// TIA Portal V17 export
// export: Created 2025-03-07T09:17:02.6439569Z, ExportSetting WithDefaults, DisplayName Totally Integrated Automation Portal, DisplayVersion V17 Update 8, DisplayName TIA Portal Openness, DisplayVersion V17 Update 8, DisplayName TIA Portal Version Control Interface, DisplayVersion V17, DisplayName SINAMICS Startdrive Advanced, DisplayVersion V17 SP2, DisplayName SINAMICS Startdrive G110M, G120, G120C, G120D, G120P, G115D, DisplayVersion V17 SP2, DisplayName SINAMICS Startdrive G130, G150, S120, S150, SINAMICS MV, S210, DisplayVersion V17 SP2, DisplayName STEP 7 Professional, DisplayVersion V17 Update 8, DisplayName SINUMERIK ONE STEP 7 Toolbox, DisplayVersion V17 Update 12, DisplayName SINUMERIK 840D sl STEP 7 Toolbox, DisplayVersion V17 Update 12, DisplayName STEP 7 Safety, DisplayVersion V17 Update 6, DisplayName WinCC Advanced, DisplayVersion V17 Update 8
FUNCTION "FC7450_QUALITY_CHECK_CLADDING" : Void   // FC7450, LAD
{ S7_Optimized_Access := 'FALSE' }
AUTHOR : ETXETAR
NAME : GM-QC
VERSION : 1.0
// stored: AutoNumber false, IsIECCheckEnabled false, SetENOAutomatically false, UDAEnableTagReadback false
BEGIN

REGION Network 1: OPTIONS OFF
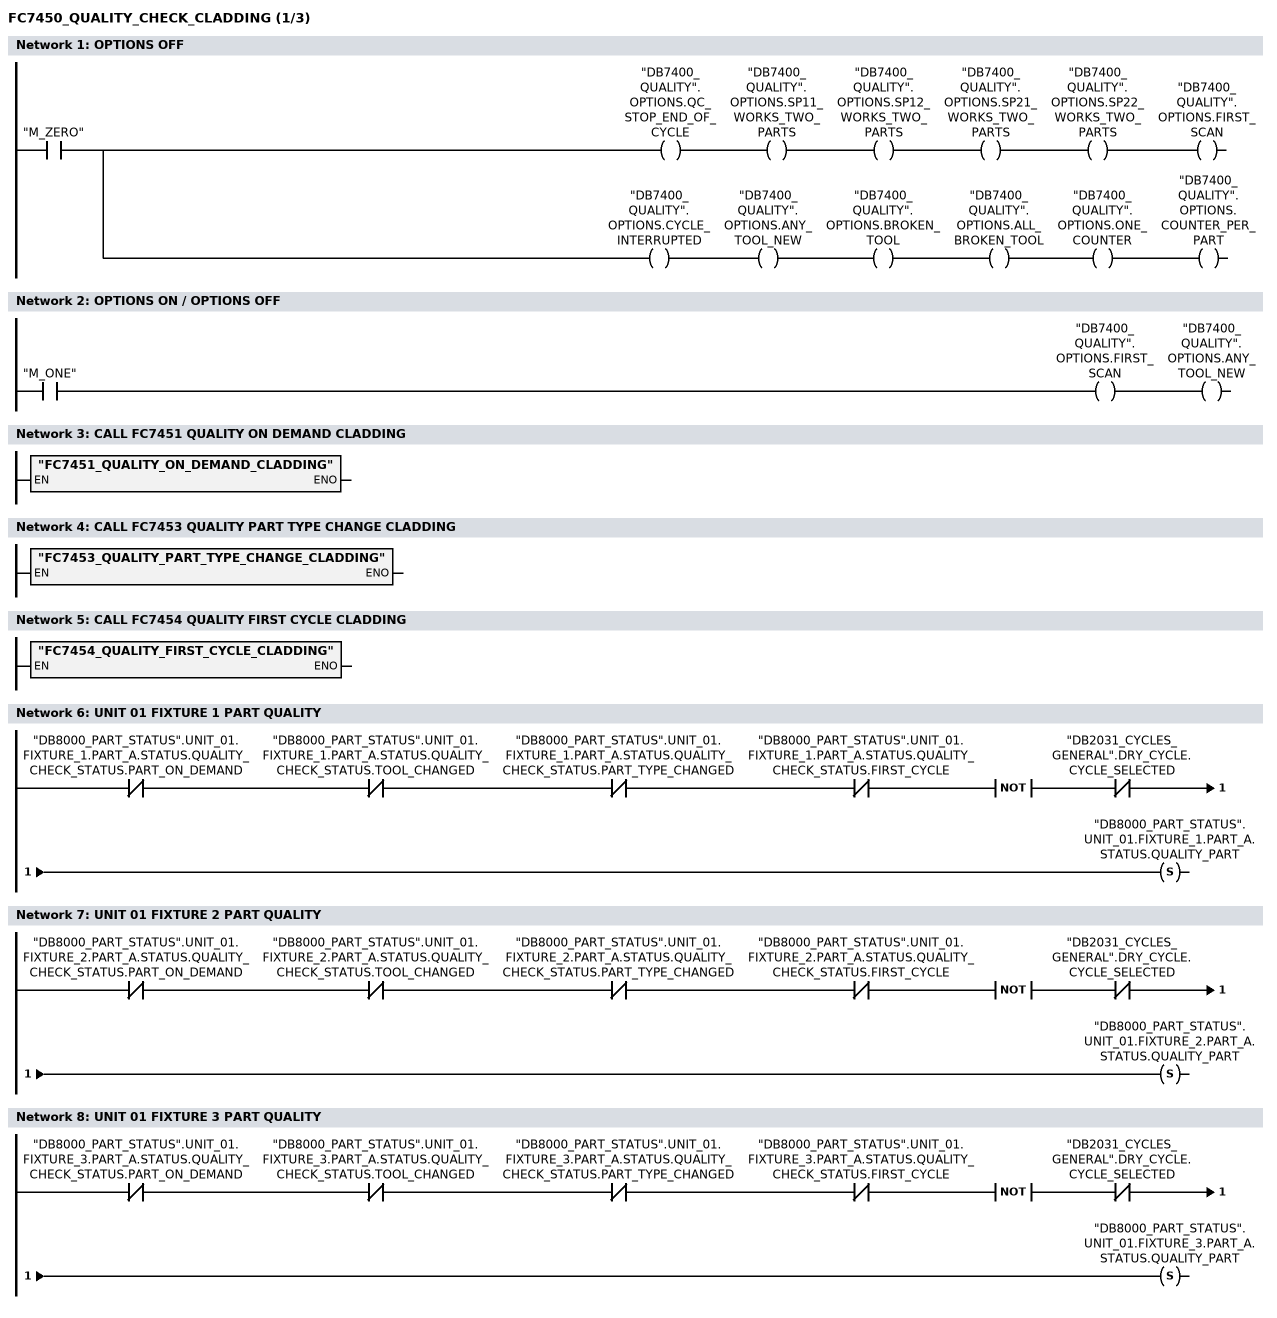
   RUNG wire#powerrail
      Contact( "M_ZERO" )
      wire#w1
      Coil( "DB7400_QUALITY".OPTIONS.QC_STOP_END_OF_CYCLE )
      Coil( "DB7400_QUALITY".OPTIONS.SP11_WORKS_TWO_PARTS )
      Coil( "DB7400_QUALITY".OPTIONS.SP12_WORKS_TWO_PARTS )
      Coil( "DB7400_QUALITY".OPTIONS.SP21_WORKS_TWO_PARTS )
      Coil( "DB7400_QUALITY".OPTIONS.SP22_WORKS_TWO_PARTS )
      Coil( "DB7400_QUALITY".OPTIONS.FIRST_SCAN )
   END_RUNG
   RUNG wire#w1
      Coil( "DB7400_QUALITY".OPTIONS.CYCLE_INTERRUPTED )
      Coil( "DB7400_QUALITY".OPTIONS.ANY_TOOL_NEW )
      Coil( "DB7400_QUALITY".OPTIONS.BROKEN_TOOL )
      Coil( "DB7400_QUALITY".OPTIONS.ALL_BROKEN_TOOL )
      Coil( "DB7400_QUALITY".OPTIONS.ONE_COUNTER )
      Coil( "DB7400_QUALITY".OPTIONS.COUNTER_PER_PART )
   END_RUNG
   // the same network as SCL:
   "DB7400_QUALITY".OPTIONS.QC_STOP_END_OF_CYCLE := "M_ZERO";
   "DB7400_QUALITY".OPTIONS.SP11_WORKS_TWO_PARTS := "M_ZERO";
   "DB7400_QUALITY".OPTIONS.SP12_WORKS_TWO_PARTS := "M_ZERO";
   "DB7400_QUALITY".OPTIONS.SP21_WORKS_TWO_PARTS := "M_ZERO";
   "DB7400_QUALITY".OPTIONS.SP22_WORKS_TWO_PARTS := "M_ZERO";
   "DB7400_QUALITY".OPTIONS.FIRST_SCAN := "M_ZERO";
   "DB7400_QUALITY".OPTIONS.CYCLE_INTERRUPTED := "M_ZERO";
   "DB7400_QUALITY".OPTIONS.ANY_TOOL_NEW := "M_ZERO";
   "DB7400_QUALITY".OPTIONS.BROKEN_TOOL := "M_ZERO";
   "DB7400_QUALITY".OPTIONS.ALL_BROKEN_TOOL := "M_ZERO";
   "DB7400_QUALITY".OPTIONS.ONE_COUNTER := "M_ZERO";
   "DB7400_QUALITY".OPTIONS.COUNTER_PER_PART := "M_ZERO";
END_REGION

REGION Network 2: OPTIONS ON / OPTIONS OFF
   RUNG wire#powerrail
      Contact( "M_ONE" )
      Coil( "DB7400_QUALITY".OPTIONS.FIRST_SCAN )
      Coil( "DB7400_QUALITY".OPTIONS.ANY_TOOL_NEW )
   END_RUNG
   // the same network as SCL:
   "DB7400_QUALITY".OPTIONS.FIRST_SCAN := "M_ONE";
   "DB7400_QUALITY".OPTIONS.ANY_TOOL_NEW := "M_ONE";
END_REGION

REGION Network 3: CALL FC7451 QUALITY ON DEMAND CLADDING
   RUNG wire#powerrail
      "FC7451_QUALITY_ON_DEMAND_CLADDING"()
   END_RUNG
   // the same network as SCL:
   "FC7451_QUALITY_ON_DEMAND_CLADDING"();
END_REGION

REGION Network 4: CALL FC7453 QUALITY PART TYPE CHANGE CLADDING
   RUNG wire#powerrail
      "FC7453_QUALITY_PART_TYPE_CHANGE_CLADDING"()
   END_RUNG
   // the same network as SCL:
   "FC7453_QUALITY_PART_TYPE_CHANGE_CLADDING"();
END_REGION

REGION Network 5: CALL FC7454 QUALITY FIRST CYCLE CLADDING
   RUNG wire#powerrail
      "FC7454_QUALITY_FIRST_CYCLE_CLADDING"()
   END_RUNG
   // the same network as SCL:
   "FC7454_QUALITY_FIRST_CYCLE_CLADDING"();
END_REGION

REGION Network 6: UNIT 01 FIXTURE 1 PART QUALITY
   RUNG wire#powerrail
      I_Contact( "DB8000_PART_STATUS".UNIT_01.FIXTURE_1.PART_A.STATUS.QUALITY_CHECK_STATUS.PART_ON_DEMAND )
      I_Contact( "DB8000_PART_STATUS".UNIT_01.FIXTURE_1.PART_A.STATUS.QUALITY_CHECK_STATUS.TOOL_CHANGED )
      I_Contact( "DB8000_PART_STATUS".UNIT_01.FIXTURE_1.PART_A.STATUS.QUALITY_CHECK_STATUS.PART_TYPE_CHANGED )
      I_Contact( "DB8000_PART_STATUS".UNIT_01.FIXTURE_1.PART_A.STATUS.QUALITY_CHECK_STATUS.FIRST_CYCLE )
      Not()
      I_Contact( "DB2031_CYCLES_GENERAL".DRY_CYCLE.CYCLE_SELECTED )
      S_Coil( "DB8000_PART_STATUS".UNIT_01.FIXTURE_1.PART_A.STATUS.QUALITY_PART )
   END_RUNG
   // the same network as SCL:
   IF NOT (NOT "DB8000_PART_STATUS".UNIT_01.FIXTURE_1.PART_A.STATUS.QUALITY_CHECK_STATUS.PART_ON_DEMAND AND NOT "DB8000_PART_STATUS".UNIT_01.FIXTURE_1.PART_A.STATUS.QUALITY_CHECK_STATUS.TOOL_CHANGED AND NOT "DB8000_PART_STATUS".UNIT_01.FIXTURE_1.PART_A.STATUS.QUALITY_CHECK_STATUS.PART_TYPE_CHANGED AND NOT "DB8000_PART_STATUS".UNIT_01.FIXTURE_1.PART_A.STATUS.QUALITY_CHECK_STATUS.FIRST_CYCLE) AND NOT "DB2031_CYCLES_GENERAL".DRY_CYCLE.CYCLE_SELECTED THEN
       "DB8000_PART_STATUS".UNIT_01.FIXTURE_1.PART_A.STATUS.QUALITY_PART := TRUE;
   END_IF;
END_REGION

REGION Network 7: UNIT 01 FIXTURE 2 PART QUALITY
   RUNG wire#powerrail
      I_Contact( "DB8000_PART_STATUS".UNIT_01.FIXTURE_2.PART_A.STATUS.QUALITY_CHECK_STATUS.PART_ON_DEMAND )
      I_Contact( "DB8000_PART_STATUS".UNIT_01.FIXTURE_2.PART_A.STATUS.QUALITY_CHECK_STATUS.TOOL_CHANGED )
      I_Contact( "DB8000_PART_STATUS".UNIT_01.FIXTURE_2.PART_A.STATUS.QUALITY_CHECK_STATUS.PART_TYPE_CHANGED )
      I_Contact( "DB8000_PART_STATUS".UNIT_01.FIXTURE_2.PART_A.STATUS.QUALITY_CHECK_STATUS.FIRST_CYCLE )
      Not()
      I_Contact( "DB2031_CYCLES_GENERAL".DRY_CYCLE.CYCLE_SELECTED )
      S_Coil( "DB8000_PART_STATUS".UNIT_01.FIXTURE_2.PART_A.STATUS.QUALITY_PART )
   END_RUNG
   // the same network as SCL:
   IF NOT (NOT "DB8000_PART_STATUS".UNIT_01.FIXTURE_2.PART_A.STATUS.QUALITY_CHECK_STATUS.PART_ON_DEMAND AND NOT "DB8000_PART_STATUS".UNIT_01.FIXTURE_2.PART_A.STATUS.QUALITY_CHECK_STATUS.TOOL_CHANGED AND NOT "DB8000_PART_STATUS".UNIT_01.FIXTURE_2.PART_A.STATUS.QUALITY_CHECK_STATUS.PART_TYPE_CHANGED AND NOT "DB8000_PART_STATUS".UNIT_01.FIXTURE_2.PART_A.STATUS.QUALITY_CHECK_STATUS.FIRST_CYCLE) AND NOT "DB2031_CYCLES_GENERAL".DRY_CYCLE.CYCLE_SELECTED THEN
       "DB8000_PART_STATUS".UNIT_01.FIXTURE_2.PART_A.STATUS.QUALITY_PART := TRUE;
   END_IF;
END_REGION

REGION Network 8: UNIT 01 FIXTURE 3 PART QUALITY
   RUNG wire#powerrail
      I_Contact( "DB8000_PART_STATUS".UNIT_01.FIXTURE_3.PART_A.STATUS.QUALITY_CHECK_STATUS.PART_ON_DEMAND )
      I_Contact( "DB8000_PART_STATUS".UNIT_01.FIXTURE_3.PART_A.STATUS.QUALITY_CHECK_STATUS.TOOL_CHANGED )
      I_Contact( "DB8000_PART_STATUS".UNIT_01.FIXTURE_3.PART_A.STATUS.QUALITY_CHECK_STATUS.PART_TYPE_CHANGED )
      I_Contact( "DB8000_PART_STATUS".UNIT_01.FIXTURE_3.PART_A.STATUS.QUALITY_CHECK_STATUS.FIRST_CYCLE )
      Not()
      I_Contact( "DB2031_CYCLES_GENERAL".DRY_CYCLE.CYCLE_SELECTED )
      S_Coil( "DB8000_PART_STATUS".UNIT_01.FIXTURE_3.PART_A.STATUS.QUALITY_PART )
   END_RUNG
   // the same network as SCL:
   IF NOT (NOT "DB8000_PART_STATUS".UNIT_01.FIXTURE_3.PART_A.STATUS.QUALITY_CHECK_STATUS.PART_ON_DEMAND AND NOT "DB8000_PART_STATUS".UNIT_01.FIXTURE_3.PART_A.STATUS.QUALITY_CHECK_STATUS.TOOL_CHANGED AND NOT "DB8000_PART_STATUS".UNIT_01.FIXTURE_3.PART_A.STATUS.QUALITY_CHECK_STATUS.PART_TYPE_CHANGED AND NOT "DB8000_PART_STATUS".UNIT_01.FIXTURE_3.PART_A.STATUS.QUALITY_CHECK_STATUS.FIRST_CYCLE) AND NOT "DB2031_CYCLES_GENERAL".DRY_CYCLE.CYCLE_SELECTED THEN
       "DB8000_PART_STATUS".UNIT_01.FIXTURE_3.PART_A.STATUS.QUALITY_PART := TRUE;
   END_IF;
END_REGION

REGION Network 9: UNIT 01 FIXTURE 4 PART QUALITY
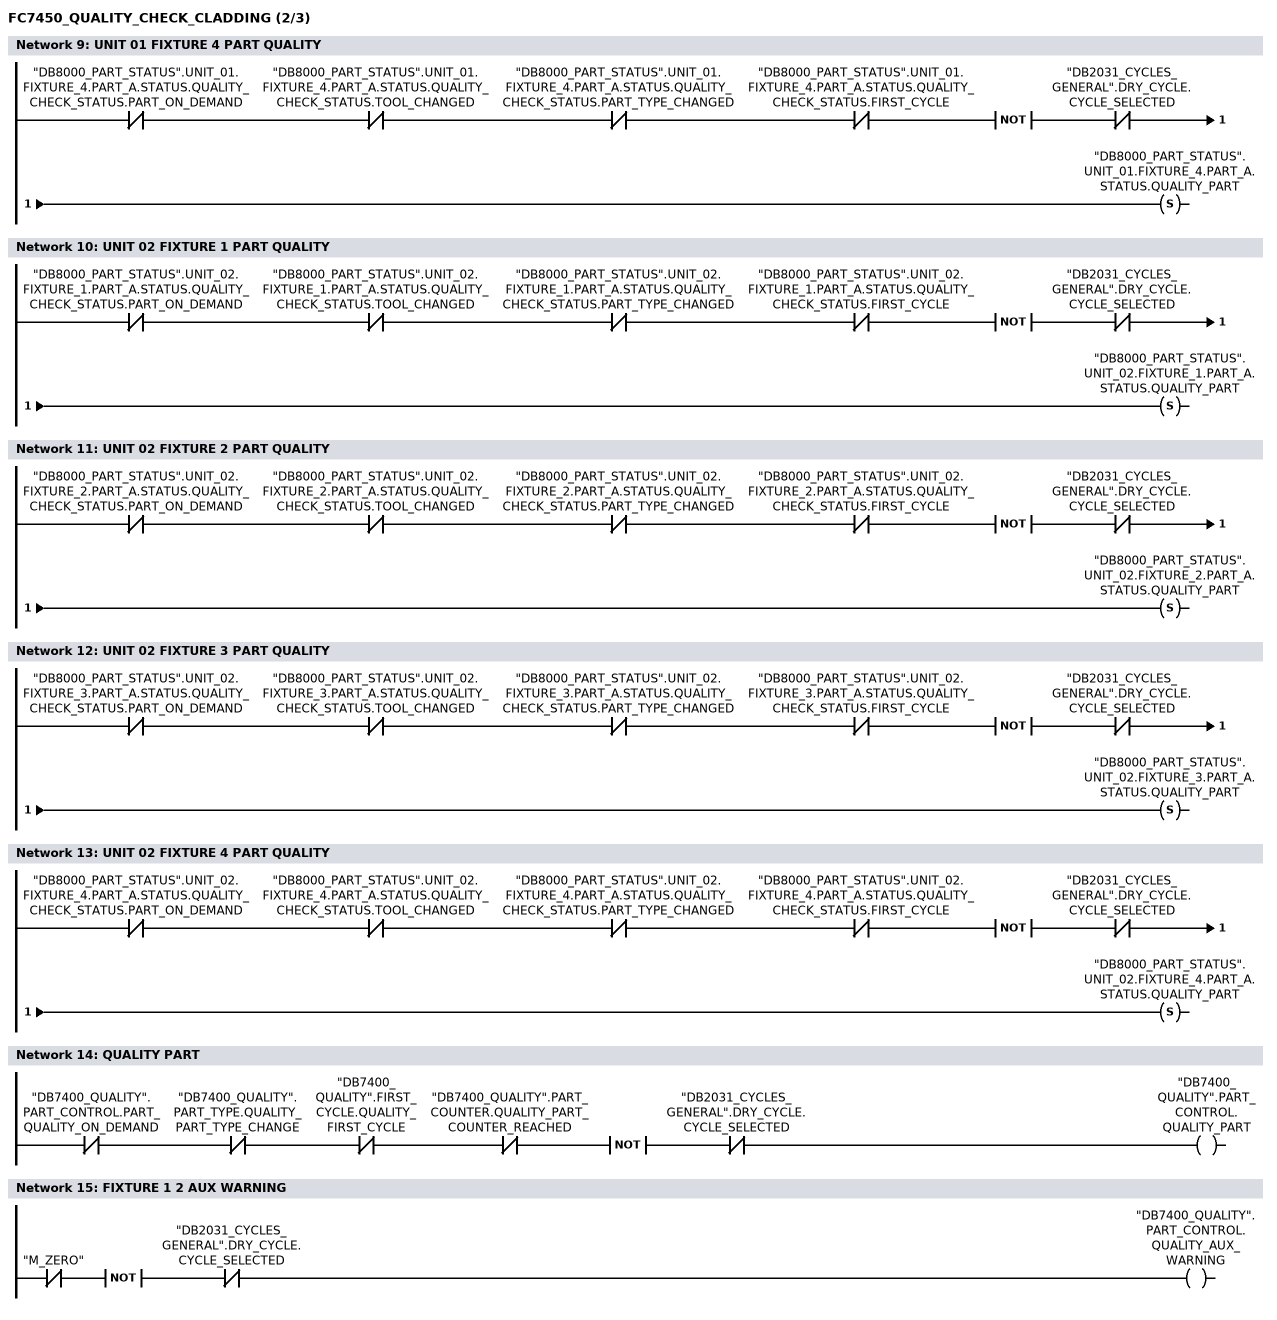
   RUNG wire#powerrail
      I_Contact( "DB8000_PART_STATUS".UNIT_01.FIXTURE_4.PART_A.STATUS.QUALITY_CHECK_STATUS.PART_ON_DEMAND )
      I_Contact( "DB8000_PART_STATUS".UNIT_01.FIXTURE_4.PART_A.STATUS.QUALITY_CHECK_STATUS.TOOL_CHANGED )
      I_Contact( "DB8000_PART_STATUS".UNIT_01.FIXTURE_4.PART_A.STATUS.QUALITY_CHECK_STATUS.PART_TYPE_CHANGED )
      I_Contact( "DB8000_PART_STATUS".UNIT_01.FIXTURE_4.PART_A.STATUS.QUALITY_CHECK_STATUS.FIRST_CYCLE )
      Not()
      I_Contact( "DB2031_CYCLES_GENERAL".DRY_CYCLE.CYCLE_SELECTED )
      S_Coil( "DB8000_PART_STATUS".UNIT_01.FIXTURE_4.PART_A.STATUS.QUALITY_PART )
   END_RUNG
   // the same network as SCL:
   IF NOT (NOT "DB8000_PART_STATUS".UNIT_01.FIXTURE_4.PART_A.STATUS.QUALITY_CHECK_STATUS.PART_ON_DEMAND AND NOT "DB8000_PART_STATUS".UNIT_01.FIXTURE_4.PART_A.STATUS.QUALITY_CHECK_STATUS.TOOL_CHANGED AND NOT "DB8000_PART_STATUS".UNIT_01.FIXTURE_4.PART_A.STATUS.QUALITY_CHECK_STATUS.PART_TYPE_CHANGED AND NOT "DB8000_PART_STATUS".UNIT_01.FIXTURE_4.PART_A.STATUS.QUALITY_CHECK_STATUS.FIRST_CYCLE) AND NOT "DB2031_CYCLES_GENERAL".DRY_CYCLE.CYCLE_SELECTED THEN
       "DB8000_PART_STATUS".UNIT_01.FIXTURE_4.PART_A.STATUS.QUALITY_PART := TRUE;
   END_IF;
END_REGION

REGION Network 10: UNIT 02 FIXTURE 1 PART QUALITY
   RUNG wire#powerrail
      I_Contact( "DB8000_PART_STATUS".UNIT_02.FIXTURE_1.PART_A.STATUS.QUALITY_CHECK_STATUS.PART_ON_DEMAND )
      I_Contact( "DB8000_PART_STATUS".UNIT_02.FIXTURE_1.PART_A.STATUS.QUALITY_CHECK_STATUS.TOOL_CHANGED )
      I_Contact( "DB8000_PART_STATUS".UNIT_02.FIXTURE_1.PART_A.STATUS.QUALITY_CHECK_STATUS.PART_TYPE_CHANGED )
      I_Contact( "DB8000_PART_STATUS".UNIT_02.FIXTURE_1.PART_A.STATUS.QUALITY_CHECK_STATUS.FIRST_CYCLE )
      Not()
      I_Contact( "DB2031_CYCLES_GENERAL".DRY_CYCLE.CYCLE_SELECTED )
      S_Coil( "DB8000_PART_STATUS".UNIT_02.FIXTURE_1.PART_A.STATUS.QUALITY_PART )
   END_RUNG
   // the same network as SCL:
   IF NOT (NOT "DB8000_PART_STATUS".UNIT_02.FIXTURE_1.PART_A.STATUS.QUALITY_CHECK_STATUS.PART_ON_DEMAND AND NOT "DB8000_PART_STATUS".UNIT_02.FIXTURE_1.PART_A.STATUS.QUALITY_CHECK_STATUS.TOOL_CHANGED AND NOT "DB8000_PART_STATUS".UNIT_02.FIXTURE_1.PART_A.STATUS.QUALITY_CHECK_STATUS.PART_TYPE_CHANGED AND NOT "DB8000_PART_STATUS".UNIT_02.FIXTURE_1.PART_A.STATUS.QUALITY_CHECK_STATUS.FIRST_CYCLE) AND NOT "DB2031_CYCLES_GENERAL".DRY_CYCLE.CYCLE_SELECTED THEN
       "DB8000_PART_STATUS".UNIT_02.FIXTURE_1.PART_A.STATUS.QUALITY_PART := TRUE;
   END_IF;
END_REGION

REGION Network 11: UNIT 02 FIXTURE 2 PART QUALITY
   RUNG wire#powerrail
      I_Contact( "DB8000_PART_STATUS".UNIT_02.FIXTURE_2.PART_A.STATUS.QUALITY_CHECK_STATUS.PART_ON_DEMAND )
      I_Contact( "DB8000_PART_STATUS".UNIT_02.FIXTURE_2.PART_A.STATUS.QUALITY_CHECK_STATUS.TOOL_CHANGED )
      I_Contact( "DB8000_PART_STATUS".UNIT_02.FIXTURE_2.PART_A.STATUS.QUALITY_CHECK_STATUS.PART_TYPE_CHANGED )
      I_Contact( "DB8000_PART_STATUS".UNIT_02.FIXTURE_2.PART_A.STATUS.QUALITY_CHECK_STATUS.FIRST_CYCLE )
      Not()
      I_Contact( "DB2031_CYCLES_GENERAL".DRY_CYCLE.CYCLE_SELECTED )
      S_Coil( "DB8000_PART_STATUS".UNIT_02.FIXTURE_2.PART_A.STATUS.QUALITY_PART )
   END_RUNG
   // the same network as SCL:
   IF NOT (NOT "DB8000_PART_STATUS".UNIT_02.FIXTURE_2.PART_A.STATUS.QUALITY_CHECK_STATUS.PART_ON_DEMAND AND NOT "DB8000_PART_STATUS".UNIT_02.FIXTURE_2.PART_A.STATUS.QUALITY_CHECK_STATUS.TOOL_CHANGED AND NOT "DB8000_PART_STATUS".UNIT_02.FIXTURE_2.PART_A.STATUS.QUALITY_CHECK_STATUS.PART_TYPE_CHANGED AND NOT "DB8000_PART_STATUS".UNIT_02.FIXTURE_2.PART_A.STATUS.QUALITY_CHECK_STATUS.FIRST_CYCLE) AND NOT "DB2031_CYCLES_GENERAL".DRY_CYCLE.CYCLE_SELECTED THEN
       "DB8000_PART_STATUS".UNIT_02.FIXTURE_2.PART_A.STATUS.QUALITY_PART := TRUE;
   END_IF;
END_REGION

REGION Network 12: UNIT 02 FIXTURE 3 PART QUALITY
   RUNG wire#powerrail
      I_Contact( "DB8000_PART_STATUS".UNIT_02.FIXTURE_3.PART_A.STATUS.QUALITY_CHECK_STATUS.PART_ON_DEMAND )
      I_Contact( "DB8000_PART_STATUS".UNIT_02.FIXTURE_3.PART_A.STATUS.QUALITY_CHECK_STATUS.TOOL_CHANGED )
      I_Contact( "DB8000_PART_STATUS".UNIT_02.FIXTURE_3.PART_A.STATUS.QUALITY_CHECK_STATUS.PART_TYPE_CHANGED )
      I_Contact( "DB8000_PART_STATUS".UNIT_02.FIXTURE_3.PART_A.STATUS.QUALITY_CHECK_STATUS.FIRST_CYCLE )
      Not()
      I_Contact( "DB2031_CYCLES_GENERAL".DRY_CYCLE.CYCLE_SELECTED )
      S_Coil( "DB8000_PART_STATUS".UNIT_02.FIXTURE_3.PART_A.STATUS.QUALITY_PART )
   END_RUNG
   // the same network as SCL:
   IF NOT (NOT "DB8000_PART_STATUS".UNIT_02.FIXTURE_3.PART_A.STATUS.QUALITY_CHECK_STATUS.PART_ON_DEMAND AND NOT "DB8000_PART_STATUS".UNIT_02.FIXTURE_3.PART_A.STATUS.QUALITY_CHECK_STATUS.TOOL_CHANGED AND NOT "DB8000_PART_STATUS".UNIT_02.FIXTURE_3.PART_A.STATUS.QUALITY_CHECK_STATUS.PART_TYPE_CHANGED AND NOT "DB8000_PART_STATUS".UNIT_02.FIXTURE_3.PART_A.STATUS.QUALITY_CHECK_STATUS.FIRST_CYCLE) AND NOT "DB2031_CYCLES_GENERAL".DRY_CYCLE.CYCLE_SELECTED THEN
       "DB8000_PART_STATUS".UNIT_02.FIXTURE_3.PART_A.STATUS.QUALITY_PART := TRUE;
   END_IF;
END_REGION

REGION Network 13: UNIT 02 FIXTURE 4 PART QUALITY
   RUNG wire#powerrail
      I_Contact( "DB8000_PART_STATUS".UNIT_02.FIXTURE_4.PART_A.STATUS.QUALITY_CHECK_STATUS.PART_ON_DEMAND )
      I_Contact( "DB8000_PART_STATUS".UNIT_02.FIXTURE_4.PART_A.STATUS.QUALITY_CHECK_STATUS.TOOL_CHANGED )
      I_Contact( "DB8000_PART_STATUS".UNIT_02.FIXTURE_4.PART_A.STATUS.QUALITY_CHECK_STATUS.PART_TYPE_CHANGED )
      I_Contact( "DB8000_PART_STATUS".UNIT_02.FIXTURE_4.PART_A.STATUS.QUALITY_CHECK_STATUS.FIRST_CYCLE )
      Not()
      I_Contact( "DB2031_CYCLES_GENERAL".DRY_CYCLE.CYCLE_SELECTED )
      S_Coil( "DB8000_PART_STATUS".UNIT_02.FIXTURE_4.PART_A.STATUS.QUALITY_PART )
   END_RUNG
   // the same network as SCL:
   IF NOT (NOT "DB8000_PART_STATUS".UNIT_02.FIXTURE_4.PART_A.STATUS.QUALITY_CHECK_STATUS.PART_ON_DEMAND AND NOT "DB8000_PART_STATUS".UNIT_02.FIXTURE_4.PART_A.STATUS.QUALITY_CHECK_STATUS.TOOL_CHANGED AND NOT "DB8000_PART_STATUS".UNIT_02.FIXTURE_4.PART_A.STATUS.QUALITY_CHECK_STATUS.PART_TYPE_CHANGED AND NOT "DB8000_PART_STATUS".UNIT_02.FIXTURE_4.PART_A.STATUS.QUALITY_CHECK_STATUS.FIRST_CYCLE) AND NOT "DB2031_CYCLES_GENERAL".DRY_CYCLE.CYCLE_SELECTED THEN
       "DB8000_PART_STATUS".UNIT_02.FIXTURE_4.PART_A.STATUS.QUALITY_PART := TRUE;
   END_IF;
END_REGION

REGION Network 14: QUALITY PART
   RUNG wire#powerrail
      I_Contact( "DB7400_QUALITY".PART_CONTROL.PART_QUALITY_ON_DEMAND )
      I_Contact( "DB7400_QUALITY".PART_TYPE.QUALITY_PART_TYPE_CHANGE )
      I_Contact( "DB7400_QUALITY".FIRST_CYCLE.QUALITY_FIRST_CYCLE )
      I_Contact( "DB7400_QUALITY".PART_COUNTER.QUALITY_PART_COUNTER_REACHED )
      Not()
      I_Contact( "DB2031_CYCLES_GENERAL".DRY_CYCLE.CYCLE_SELECTED )
      Coil( "DB7400_QUALITY".PART_CONTROL.QUALITY_PART )
   END_RUNG
   // the same network as SCL:
   "DB7400_QUALITY".PART_CONTROL.QUALITY_PART := NOT (NOT "DB7400_QUALITY".PART_CONTROL.PART_QUALITY_ON_DEMAND AND NOT "DB7400_QUALITY".PART_TYPE.QUALITY_PART_TYPE_CHANGE AND NOT "DB7400_QUALITY".FIRST_CYCLE.QUALITY_FIRST_CYCLE AND NOT "DB7400_QUALITY".PART_COUNTER.QUALITY_PART_COUNTER_REACHED) AND NOT "DB2031_CYCLES_GENERAL".DRY_CYCLE.CYCLE_SELECTED;
END_REGION

REGION Network 15: FIXTURE 1 2 AUX WARNING
   RUNG wire#powerrail
      I_Contact( "M_ZERO" )
      Not()
      I_Contact( "DB2031_CYCLES_GENERAL".DRY_CYCLE.CYCLE_SELECTED )
      Coil( "DB7400_QUALITY".PART_CONTROL.QUALITY_AUX_WARNING )
   END_RUNG
   // the same network as SCL:
   "DB7400_QUALITY".PART_CONTROL.QUALITY_AUX_WARNING := NOT (NOT "M_ZERO") AND NOT "DB2031_CYCLES_GENERAL".DRY_CYCLE.CYCLE_SELECTED;
END_REGION

REGION Network 16: FIXTURE 1 2 AUX FAULT
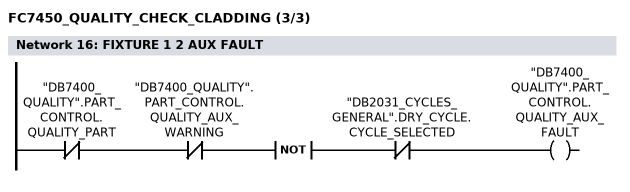
   RUNG wire#powerrail
      I_Contact( "DB7400_QUALITY".PART_CONTROL.QUALITY_PART )
      I_Contact( "DB7400_QUALITY".PART_CONTROL.QUALITY_AUX_WARNING )
      Not()
      I_Contact( "DB2031_CYCLES_GENERAL".DRY_CYCLE.CYCLE_SELECTED )
      Coil( "DB7400_QUALITY".PART_CONTROL.QUALITY_AUX_FAULT )
   END_RUNG
   // the same network as SCL:
   "DB7400_QUALITY".PART_CONTROL.QUALITY_AUX_FAULT := NOT (NOT "DB7400_QUALITY".PART_CONTROL.QUALITY_PART AND NOT "DB7400_QUALITY".PART_CONTROL.QUALITY_AUX_WARNING) AND NOT "DB2031_CYCLES_GENERAL".DRY_CYCLE.CYCLE_SELECTED;
END_REGION
END_FUNCTION
